{attribute 'linkalways'} 
{attribute 'no_explicit_call' := 'This FB is a CLASS and must be accessed using methods or properties'}
{attribute 'enable_dynamic_creation'}
FUNCTION_BLOCK Node_F_VN_AddToContainerElements_REAL EXTENDS VisionNode
VAR
    fValue : _REAL(0.0);
    ipContainer : _ITcVnContainer;
    hrPrev : _HRESULT(S_OK);
    hresult : _HRESULT(S_OK);
END_VAR

METHOD PUBLIC  Clone : I_Node
VAR
    pNode : POINTER TO Node_F_VN_AddToContainerElements_REAL;
END_VAR
pNode := __NEW(Node_F_VN_AddToContainerElements_REAL);
Clone := pNode^;
END_METHOD

METHOD FB_init : BOOL
VAR_INPUT
    bInitRetains : BOOL; // if TRUE, the retain variables are initialized (warm start / cold start)
    bInCopyCode : BOOL;  // if TRUE, the instance afterwards gets moved into the copy code (online change)
END_VAR
AddParameter('fValue', fValue);
AddInput('ipContainer', ipContainer);
AddInput('hrPrev', hrPrev);
AddOutput('ipContainer', ipContainer);
AddOutput('hresult',hresult);
END_METHOD

METHOD PROTECTED OnExecute
hresult.Value := F_VN_AddToContainerElements_REAL(
    fValue := fValue.Value,
    ipContainer := ipContainer.Value,
    hrPrev:= hrPrev.Value);
END_METHOD

METHOD PUBLIC PreExecutionCheck
VAR_INPUT
    Check : I_PreExecutionChecks;
END_VAR
Check.IsTrue(ipContainer.IsValid, 'ipContainer must be a valid container');
Check.IsTrue(ipContainer.IsType(TC_GLOBAL_CONST_LIST.ContainerType_Vector_REAL), 'ipContainer contains incorrect type');
END_METHOD

END_FUNCTION_BLOCK

(* stored: Version 1.1.0.1, ProductVersion 3.1.4026.13
   POU Node_F_VN_AddToContainerElements_REAL: Id {fb025afe-798c-4026-856d-d231b4ff62c2}, SpecialFunc None
   Folder Constructor: Id {e204f69e-ed4b-4469-9d64-612d1fbaac81}
   Method Clone: Id {b368c7eb-e662-42ef-a812-0b9c6d1e0439}
   Method FB_init: Id {4e867a8c-aac7-44c4-be64-cbcb854aa7a3}
   Method OnExecute: Id {4df75fcb-7563-4586-9f81-18b19b997ca1}
   Method PreExecutionCheck: Id {37f8a098-747c-49ff-9697-2f6446c02766} *)
